Fanuc KAREL source: kb00009.KL

-- PROVISIONAL review KL for V940-1; original PC SHA256 f23568e631a1178a2a9aa17f0b39bd3ff1edee9bdf22c9ee0220dcbb7f3a62fa
-- Incomplete behavior may be omitted. Consult companion uncertainty JSON. Do not deploy.
PROGRAM KB00009
%NOLOCKGROUP
VAR
  P1 : REAL
  P2 : REAL
  RESULT : REAL
BEGIN
  -- V9_ZERO_TABLE_METADATA_HINT layout=0001; no indexed target words; source/name/runtime held
  -- UNRESOLVED_PC offsets 5-16; opcodes 2E,23
  -- UNRESOLVED_PC offsets 21-32; opcodes 2E,23
  -- UNRESOLVED_PC offsets 37-58; opcodes 27,22,22,76,23
  -- UNRESOLVED_PC offsets 63-67; opcodes 7F
END KB00009
